(* Logix 5000 project; controller PLC2_Project_7_SensorCalibration Emulate 5570 rev 20.11; software revision 20.00 *)

TASK MainTask (continuous, watchdog 500 ms) : MainProgram

MODULES
   Local : Emulate 5570 (ICP 1, rev 20.11)
END_MODULES

ADD_ON_INSTRUCTION NSCP   (* revision 1.0 *)
// Nicks Scale With Parameters
VAR_INPUT
   InputMax : DINT; {required}
   InputMin : DINT; {required}
   ScaledMaxOut : DINT; {required}
   ScaledMinOut : DINT; {required}
   Input : DINT; {required}
END_VAR
VAR_OUTPUT
   ScaledOutput : REAL; {access Read Only, required}
END_VAR
VAR
   Rate : REAL; {access None}
END_VAR

ROUTINE Logic   (* structured text *)
   IF (EnableIn) THEN
   	Rate := (ScaledMaxOut - ScaledMinOut) / (InputMax - InputMin);
   	ScaledOutput := (Input - InputMin) * Rate + ScaledMinOut;
   END_IF;
END_ROUTINE
END_ADD_ON_INSTRUCTION

ADD_ON_INSTRUCTION SCP   (* revision 1.2, vendor Rockwell Automation *)
// Scale w/Parameters
// Help:
// Use this instruction to scale data from your analog module and bring it into the limits prescribed by the process variable or another analog module.
// Equations used in calculating a linear relationship:
// Scaled value = (input value - input min.) x rate + scaled minimum
// Rate = (scaled max. - scaled min.) / (input max. - input min.)
VAR_INPUT
   Input : REAL; {required}
   Input_Min : REAL; {required}
   Input_Max : REAL; {required}
   Scaled_Min : REAL; {required}
   Scaled_Max : REAL; {required}
END_VAR
VAR_OUTPUT
   Output : REAL; {access Read Only, required}
END_VAR
VAR
   Rate : REAL;
END_VAR

ROUTINE Logic   (* ladder *)
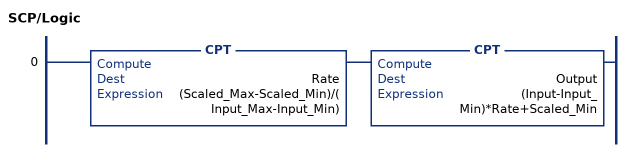
   0: CPT(Rate,(Scaled_Max-Scaled_Min)/(Input_Max-Input_Min))CPT(Output,(Input-Input_Min)*Rate+Scaled_Min);
END_ROUTINE
END_ADD_ON_INSTRUCTION

PROGRAM MainProgram   (* main routine _00_MainRoutine *)
VAR
   NSCP_O2SensorOutput : NSCP; {access Read Only}
   O2Sensor_Reading : REAL; {access Read Only}
   sim_outputSensor : REAL; {access Read Only}
   sim_oxygenGasValveInput : BOOL; {access Read Only}
   sim_timer : TIMER; {access Read Only}
   sim_zeroGasValveInput : BOOL; {access Read Only}
   Valve_TestGas_En : BOOL; {access Read Only}
   Valve_ZeroGas_En : BOOL; {access Read Only}
END_VAR

ROUTINE _00_MainRoutine   (* ladder *)
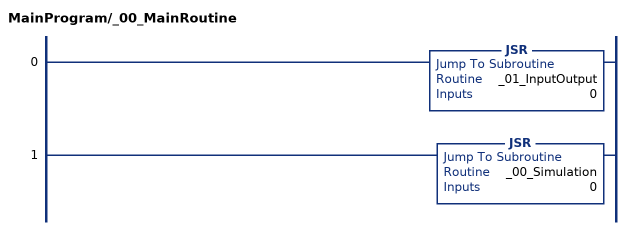
   0: JSR(_01_InputOutput,0);
   1: JSR(_00_Simulation,0);
END_ROUTINE

ROUTINE _00_Simulation   (* structured text *)
   // Analog output simulation
   // Range:
   // 0 - 16383
   // 0% - 40%
   
   IF(sim_zeroGasValveInput)THEN
   	sim_outputSensor := 0; // 0 - 16384
   END_IF;
   
   IF(sim_oxygenGasValveInput)THEN
   	sim_outputSensor := 12287; //12287 =~ 30% gas
   	//Change this value (lower) to see if the calibration works
   END_IF;
   
   //Decrease the sensor output over time to represent the sensor degrading:
   
   
   
END_ROUTINE

ROUTINE _01_InputOutput   (* ladder *)
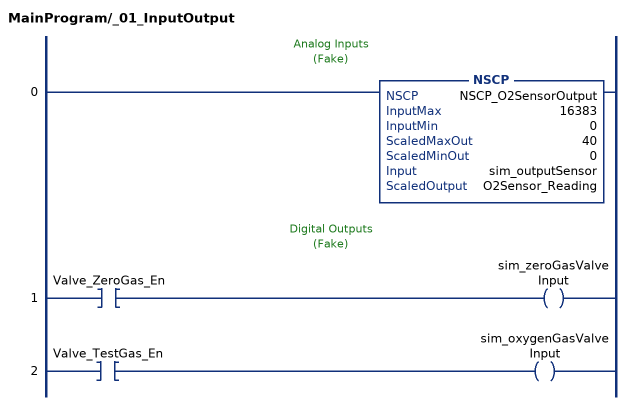
   // Analog Inputs
   // (Fake)
   0: NSCP(NSCP_O2SensorOutput,16383,0,40,0,sim_outputSensor,O2Sensor_Reading);
   // Digital Outputs
   // (Fake)
   1: XIC(Valve_ZeroGas_En)OTE(sim_zeroGasValveInput);
   2: XIC(Valve_TestGas_En)OTE(sim_oxygenGasValveInput);
END_ROUTINE
END_PROGRAM
